PROGRAM MAIN
VAR
END_VAR

HorAxisPosCon();

END_PROGRAM

(* stored: Version 1.1.0.1, ProductVersion 3.1.4024.6
   POU MAIN: Id {b2972736-a71e-42a4-967e-56ec8f4bb8c0}, SpecialFunc None *)
